# EPICS autosave request: CARSApp/Db/smartControl_settings.req
# FILE... smartControl_settings.req
$(P)$(R)debugLevel
file "smartControl_settings_axisN", P=$(P), R=$(R), AXIS=TTH
file "smartControl_settings_axisN", P=$(P), R=$(R), AXIS=OMEGA
file "smartControl_settings_axisN", P=$(P), R=$(R), AXIS=PHI
file "smartControl_settings_axisN", P=$(P), R=$(R), AXIS=KAPPA
